// TIA Portal V20 export
DATA_BLOCK "SBK13"   // DB327
// stored: MemoryReserve 100
   VAR
      SPARE_5 : Bool := FALSE;
      SPARE_6 : Bool := FALSE;
      SPARE_7 : Bool := FALSE;
      SPARE : Bool := FALSE;
      SPARE_1 : Bool := FALSE;
      SPARE_2 : Bool := FALSE;
      SPARE_3 : Bool := FALSE;
      SPARE_4 : Bool := FALSE;
      SPARE_8 : Bool := FALSE;
      SPARE_9 : Bool := FALSE;
      SPARE_10 : Bool := FALSE;
   END_VAR
BEGIN
END_DATA_BLOCK
